# EPICS autosave request: iocBoot/ioc13MeasCompETC_2/auto_settings.req
file "ETC_settings.req", P=$(P)
file "pid_control_settings.req"  P=$(P), PID=PID1
